// TIA Portal V19 export
DATA_BLOCK "Main_DB"   // DB2
{ S7_Optimized_Access := 'TRUE' }
// stored: MemoryReserve 100
   VAR
      start : Bool;
      data : String := '{"id":"3","name":"bart","age":"25"}';
      url : String := 'http://192.168.97.10:5555/users/';
      connected { ExternalWritable := 'False'} : Bool;
      done { ExternalWritable := 'False'} : Bool;
      busy { ExternalWritable := 'False'} : Bool;
      error { ExternalWritable := 'False'} : Bool;
      status { ExternalWritable := 'False'} : Word;
      response { ExternalWritable := 'False'} : Array[0..2000] of Char;
      extracted_string { S7_SetPoint := 'True'} : String;
      Return_value : Word;
      LED_1 : Bool;
      LED_2 : Bool;
      Return_value_2 : DInt;
      reset : Bool;
      blok_1_error : Bool;
   END_VAR
BEGIN
END_DATA_BLOCK
